// TIA Portal V16 export
// export: Created 2023-03-29T11:03:19.0500739Z, ExportSetting WithDefaults, DisplayName Totally Integrated Automation Portal, DisplayVersion V16 Update 6, DisplayName TIA Portal Version Control Interface, DisplayVersion V16 Update 2, DisplayName TIA Portal Openness, DisplayVersion V16 Update 6, DisplayName STEP 7 Professional, DisplayVersion V16 Update 6, DisplayName STEP 7 Safety, DisplayVersion V16, DisplayName WinCC Advanced, DisplayVersion V16 Update 6
FUNCTION "RTC" : Void   // FC44, LAD
{ S7_Optimized_Access := 'TRUE' }
VERSION : 0.1
// stored: AutoNumber true, IsIECCheckEnabled false, SetENOAutomatically false, UDAEnableTagReadback false
   VAR_TEMP   // added for the SCL form of the ladder/FBD networks
      _w1 : Bool;
      _w2 : Bool;
   END_VAR
BEGIN

REGION Network 1
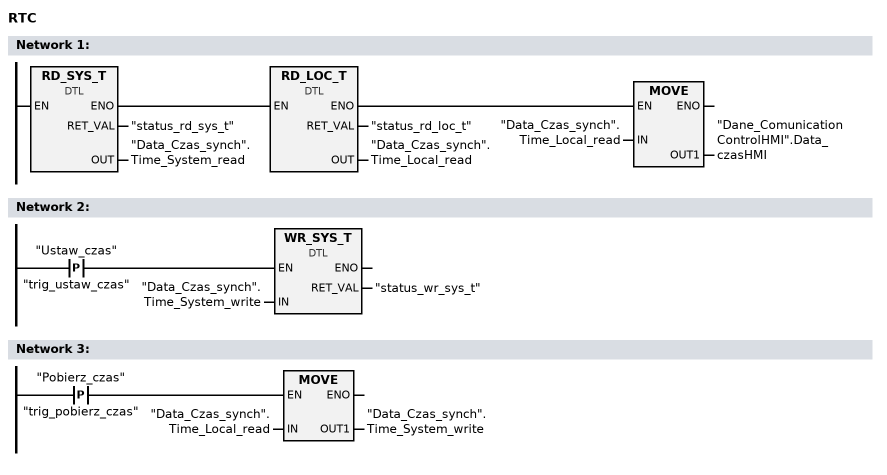
   RUNG wire#powerrail
      { S7_Templates := "date_type := DTL" } RD_SYS_T(RET_VAL => "status_rd_sys_t", OUT => "Data_Czas_synch".Time_System_read)
      { S7_Templates := "date_type := DTL" } RD_LOC_T(RET_VAL => "status_rd_loc_t", OUT => "Data_Czas_synch".Time_Local_read)
      { S7_GenerateENO := "TRUE" } Move(in := "Data_Czas_synch".Time_Local_read, out1 => "Dane_ComunicationControlHMI".Data_czasHMI)
   END_RUNG
   // the same network as SCL:
   "status_rd_sys_t" := RD_SYS_T(OUT => "Data_Czas_synch".Time_System_read, ENO => #_w1);
   "status_rd_loc_t" := RD_LOC_T(EN := #_w1, OUT => "Data_Czas_synch".Time_Local_read, ENO => #_w2);
   IF #_w2 THEN "Dane_ComunicationControlHMI".Data_czasHMI := "Data_Czas_synch".Time_Local_read; END_IF;
END_REGION

REGION Network 2
   RUNG wire#powerrail
      P_Contact(operand := "Ustaw_czas", bit := "trig_ustaw_czas")
      { S7_Templates := "date_type := DTL" } WR_SYS_T(IN := "Data_Czas_synch".Time_System_write, RET_VAL => "status_wr_sys_t")
   END_RUNG
   // the same network as SCL:
   #_w1 := "Ustaw_czas" AND NOT "trig_ustaw_czas";   // rising edge of "Ustaw_czas"
   "trig_ustaw_czas" := "Ustaw_czas";
   IF #_w1 THEN "status_wr_sys_t" := WR_SYS_T(IN := "Data_Czas_synch".Time_System_write); END_IF;
END_REGION

REGION Network 3
   RUNG wire#powerrail
      P_Contact(operand := "Pobierz_czas", bit := "trig_pobierz_czas")
      { S7_GenerateENO := "TRUE" } Move(in := "Data_Czas_synch".Time_Local_read, out1 => "Data_Czas_synch".Time_System_write)
   END_RUNG
   // the same network as SCL:
   #_w1 := "Pobierz_czas" AND NOT "trig_pobierz_czas";   // rising edge of "Pobierz_czas"
   "trig_pobierz_czas" := "Pobierz_czas";
   IF #_w1 THEN "Data_Czas_synch".Time_System_write := "Data_Czas_synch".Time_Local_read; END_IF;
END_REGION
END_FUNCTION
